TYPE st_BMS_Set :
STRUCT
	b_EnableBMS				:	BOOL;
	b_HVDC_Required			: 	BOOL;
END_STRUCT
END_TYPE

(* stored: Version 1.1.0.1, ProductVersion 3.1.4024.12
   DUT st_BMS_Set: Id {3fd25b3f-b1d6-4864-975a-be010efb693e} *)
